INTERFACE I_SimpleLogger EXTENDS I_Base

METHOD LogMessage
VAR_INPUT
	Source	: I_SimpleLogSource;
	Message : I_SimpleLogMessage;
END_VAR
END_METHOD

END_INTERFACE

(* stored: Version 1.1.0.1
   Itf I_SimpleLogger: Id {c8a1792f-cb2f-48d0-9dfa-5ceb9552924e}
   Method LogMessage: Id {0342aa65-e9de-4e01-8c5d-24488fff3663} *)
